(* IEC 61131-3 sources: CodesysTest/alpha/export/Pro18_1174.dev/Plc Logic/Application/Event Handlers, 1 file *)

(* ---- OnlineChangeDone.pou.st ---- *)
(*#-#-#-#-#-#-#-#-#-#---Declaration---#-#-#-#-#-#-#-#-#-#-#-#-#*)

FUNCTION OnlineChangeDone : DWORD
VAR_IN_OUT
	EventPrm: CmpApp.EVTPARAM_CmpApp;
END_VAR
VAR
END_VAR
(*#-#-#-#-#-#-#-#-#-#---Implementation---#-#-#-#-#-#-#-#-#-#-#-#-#*)

RecallValues();
